PROGRAM MAIN
VAR
END_VAR

END_PROGRAM

(* stored: Version 1.1.0.1
   POU MAIN: Id {89f4f3f1-64e1-4905-89d1-81ed249f636b} *)
